// TIA Portal V20 export
FUNCTION "FC_ManualSorter" : Void   // FC18, LAD
// stored: Access Published, Namespace Global, SetENOAutomatically false
   VAR_INPUT
      RunWheels : Bool;
      "GoRight/left" : Bool;
      GoStraight : Bool;
      "positionRight/Left" : Bool;
      positionStraight : Bool;
   END_VAR
   VAR_OUTPUT
      CmdRunWheels : Bool;
      "CmdRight/Left" : Bool;
      CmdStraight : Bool;
   END_VAR
BEGIN

REGION Network 1: status manual
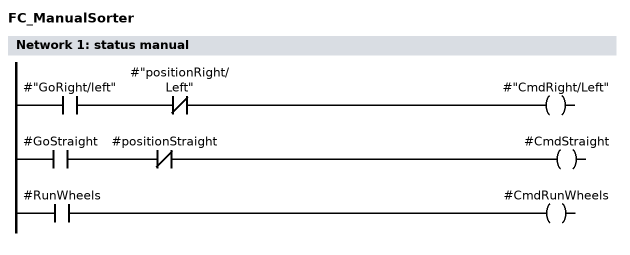
   RUNG wire#powerrail
      Contact( #"GoRight/left" )
      I_Contact( #"positionRight/Left" )
      Coil( #"CmdRight/Left" )
   END_RUNG
   RUNG wire#powerrail
      Contact( #GoStraight )
      I_Contact( #positionStraight )
      Coil( #CmdStraight )
   END_RUNG
   RUNG wire#powerrail
      Contact( #RunWheels )
      Coil( #CmdRunWheels )
   END_RUNG
   // the same network as SCL:
   #"CmdRight/Left" := #"GoRight/left" AND NOT #"positionRight/Left";
   #CmdStraight := #GoStraight AND NOT #positionStraight;
   #CmdRunWheels := #RunWheels;
END_REGION
END_FUNCTION
